FUNCTION_BLOCK UT_AuxiliaryInputMapping_Type_06_DualBool_BothNonLatched (* Type 6 DualBool_BothNonLatched Three-position switch - return to centre *)
  (* Standard: ISO 11783-6; Classification: AUX – ISO 11783-6; Function: All Inputs; Type: UT according to ISO 11783-6; Description: - Type 6 DualBool_BothNonLatched Three-position switch - return to centre Applicable AUX-N only * Maps to IX *)
  (* Version 1.0, 2018-12-05, Jose Cabral *)
  (* Version 1.1, 2022-08-04, Franz Höpfinger, HR Agrartechnik GmbH *)
  (* Version 1.2, 2023-01-05, Franz Höpfinger, HR Agrartechnik GmbH *)
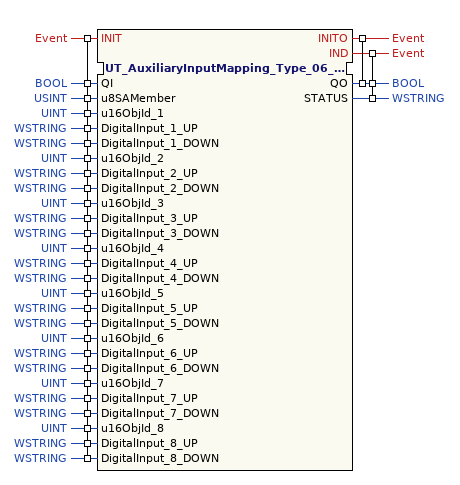
  EVENT_INPUT
    INIT WITH QI, u8SAMember, u16ObjId_1, DigitalInput_1_UP, DigitalInput_1_DOWN, u16ObjId_2, DigitalInput_2_UP, DigitalInput_2_DOWN, u16ObjId_3, DigitalInput_3_UP, DigitalInput_3_DOWN, u16ObjId_4, DigitalInput_4_UP, DigitalInput_4_DOWN, u16ObjId_5, DigitalInput_5_UP, DigitalInput_5_DOWN, u16ObjId_6, DigitalInput_6_UP, DigitalInput_6_DOWN, u16ObjId_7, DigitalInput_7_UP, DigitalInput_7_DOWN, u16ObjId_8, DigitalInput_8_UP, DigitalInput_8_DOWN; (* Service Initialization *)
  END_EVENT
  EVENT_OUTPUT
    INITO WITH QO; (* Initialization Confirm *)
    IND WITH QO, STATUS; (* Indication from Resource *)
  END_EVENT
  VAR_INPUT
    QI : BOOL; (* Event Input Qualifier *)
    u8SAMember : USINT := 255; (* Dummy !, set to 255 if in doubt. 0 deactivates FB. *)
    u16ObjId_1 : UINT := 31000; (* Object ID of Input 1 *)
    DigitalInput_1_UP : WSTRING := "AuxInput_31000_UP"; (* Identifier for Input 1 UP *)
    DigitalInput_1_DOWN : WSTRING := "AuxInput_31000_DOWN"; (* Identifier for Input 1 DOWN *)
    u16ObjId_2 : UINT := 31001; (* Object ID of Input 2 *)
    DigitalInput_2_UP : WSTRING := "AuxInput_31001_UP"; (* Identifier for Input 2 UP *)
    DigitalInput_2_DOWN : WSTRING := "AuxInput_31001_DOWN"; (* Identifier for Input 2 DOWN *)
    u16ObjId_3 : UINT := 31002; (* Object ID of Input 3 *)
    DigitalInput_3_UP : WSTRING := "AuxInput_31002_UP"; (* Identifier for Input 3 UP *)
    DigitalInput_3_DOWN : WSTRING := "AuxInput_31002_DOWN"; (* Identifier for Input 3 DOWN *)
    u16ObjId_4 : UINT := 31003; (* Object ID of Input 4 *)
    DigitalInput_4_UP : WSTRING := "AuxInput_31003_UP"; (* Identifier for Input 4 UP *)
    DigitalInput_4_DOWN : WSTRING := "AuxInput_31003_DOWN"; (* Identifier for Input 4 DOWN *)
    u16ObjId_5 : UINT := 31004; (* Object ID of Input 5 *)
    DigitalInput_5_UP : WSTRING := "AuxInput_31004_UP"; (* Identifier for Input 5 UP *)
    DigitalInput_5_DOWN : WSTRING := "AuxInput_31004_DOWN"; (* Identifier for Input 5 DOWN *)
    u16ObjId_6 : UINT := 31005; (* Object ID of Input 6 *)
    DigitalInput_6_UP : WSTRING := "AuxInput_31005_UP"; (* Identifier for Input 6 UP *)
    DigitalInput_6_DOWN : WSTRING := "AuxInput_31005_DOWN"; (* Identifier for Input 6 DOWN *)
    u16ObjId_7 : UINT := 31006; (* Object ID of Input 7 *)
    DigitalInput_7_UP : WSTRING := "AuxInput_31006_UP"; (* Identifier for Input 7 UP *)
    DigitalInput_7_DOWN : WSTRING := "AuxInput_31006_DOWN"; (* Identifier for Input 7 DOWN *)
    u16ObjId_8 : UINT := 31007; (* Object ID of Input 8 *)
    DigitalInput_8_UP : WSTRING := "AuxInput_31007_UP"; (* Identifier for Input 8 UP *)
    DigitalInput_8_DOWN : WSTRING := "AuxInput_31007_DOWN"; (* Identifier for Input 8 DOWN *)
  END_VAR
  VAR_OUTPUT
    QO : BOOL; (* Event Output Qualifier *)
    STATUS : WSTRING; (* Service Status *)
  END_VAR
END_FUNCTION_BLOCK
